% RSLogix 500 project FINAL PLC COMPLETE.RSS, saved by version 8.10.00.30 %
PROJECT "UNTITLED"    % processor: MicroLogix 1000 %

PROGRAM FILES
  LAD 2 "MAIN_PROG"  22 rungs
  LAD 3 "USER_FAULT"  1 rungs
  LAD 4 "HSC_INT"  1 rungs
  LAD 5 "STI_INT"  1 rungs
  LAD 6, 7, 8, 9, 10, 11, 12, 13, 14, 15, 16: only END

DATA FILES
  O0 OUTPUT  1 elements
  I1 INPUT  2 elements
  S2 STATUS  33 elements
  B3 BINARY  32 elements
  T4 TIMER  40 elements
  C5 COUNTER  32 elements
  R6 CONTROL  16 elements
  N7 INTEGER  105 elements

LADDER 2 "MAIN_PROG"
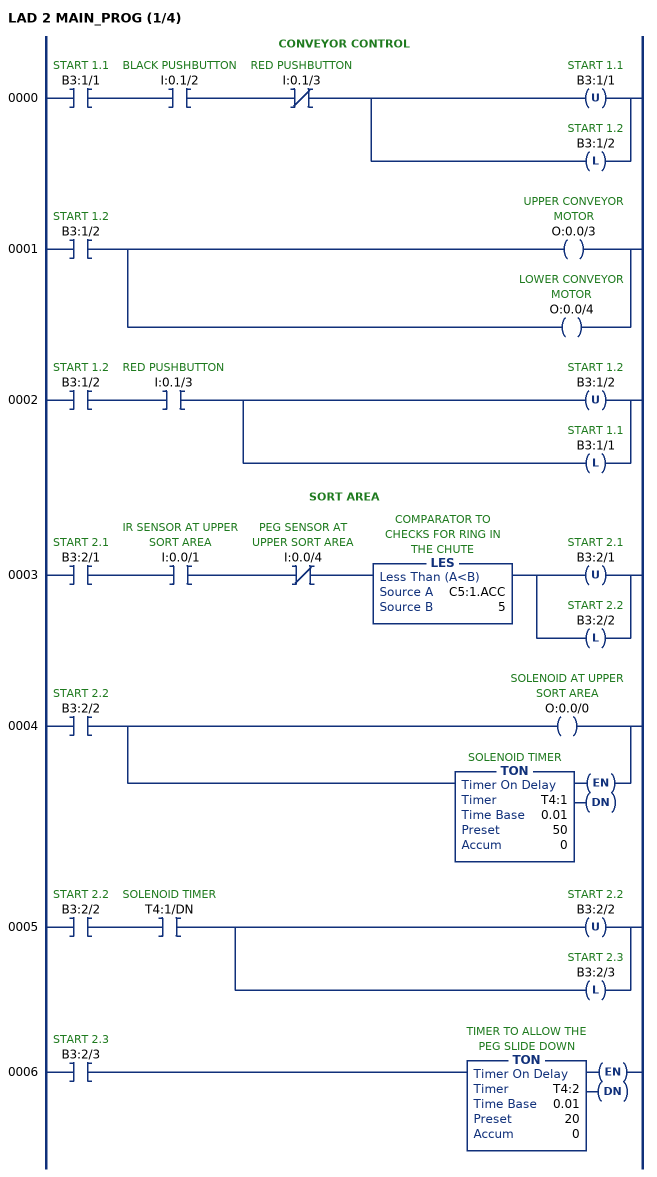
% Rung: 0 %
% TITLE: CONVEYOR CONTROL %
SOR XIC B3:1/1 XIC I:0.1/2 XIO I:0.1/3 BST OTU B3:1/1 NXB OTL B3:1/2 BND EOR
%   B3:1/1  "START 1.1" %
%   I:0.1/2  "BLACK PUSHBUTTON" %
%   I:0.1/3  "RED PUSHBUTTON" %
%   B3:1/2  "START 1.2" %
% Rung: 1 %
SOR XIC B3:1/2 BST OTE O:0.0/3 NXB OTE O:0.0/4 BND EOR
%   B3:1/2  "START 1.2" %
%   O:0.0/3  "UPPER CONVEYOR MOTOR" %
%   O:0.0/4  "LOWER CONVEYOR MOTOR" %
% Rung: 2 %
SOR XIC B3:1/2 XIC I:0.1/3 BST OTU B3:1/2 NXB OTL B3:1/1 BND EOR
%   B3:1/2  "START 1.2" %
%   I:0.1/3  "RED PUSHBUTTON" %
%   B3:1/1  "START 1.1" %
% Rung: 3 %
% TITLE: SORT AREA %
SOR XIC B3:2/1 XIC I:0.0/1 XIO I:0.0/4 LES C5:1.ACC 5 BST OTU B3:2/1 NXB OTL B3:2/2 BND EOR
%   B3:2/1  "START 2.1" %
%   I:0.0/1  "IR SENSOR AT UPPER SORT AREA" %
%   I:0.0/4  "PEG SENSOR AT UPPER SORT AREA" %
%   C5:1.ACC  "COMPARATOR TO CHECKS FOR RING IN THE CHUTE" %
%   B3:2/2  "START 2.2" %
% Rung: 4 %
SOR XIC B3:2/2 BST OTE O:0.0/0 NXB TON T4:1 0.01 50 0 BND EOR
%   B3:2/2  "START 2.2" %
%   O:0.0/0  "SOLENOID AT UPPER SORT AREA" %
%   T4:1  "SOLENOID TIMER" %
% Rung: 5 %
SOR XIC B3:2/2 XIC T4:1/DN BST OTU B3:2/2 NXB OTL B3:2/3 BND EOR
%   B3:2/2  "START 2.2" %
%   T4:1  "SOLENOID TIMER" %
%   B3:2/3  "START 2.3" %
% Rung: 6 %
SOR XIC B3:2/3 TON T4:2 0.01 20 0 EOR
%   B3:2/3  "START 2.3" %
%   T4:2  "TIMER TO ALLOW THE PEG SLIDE DOWN" %

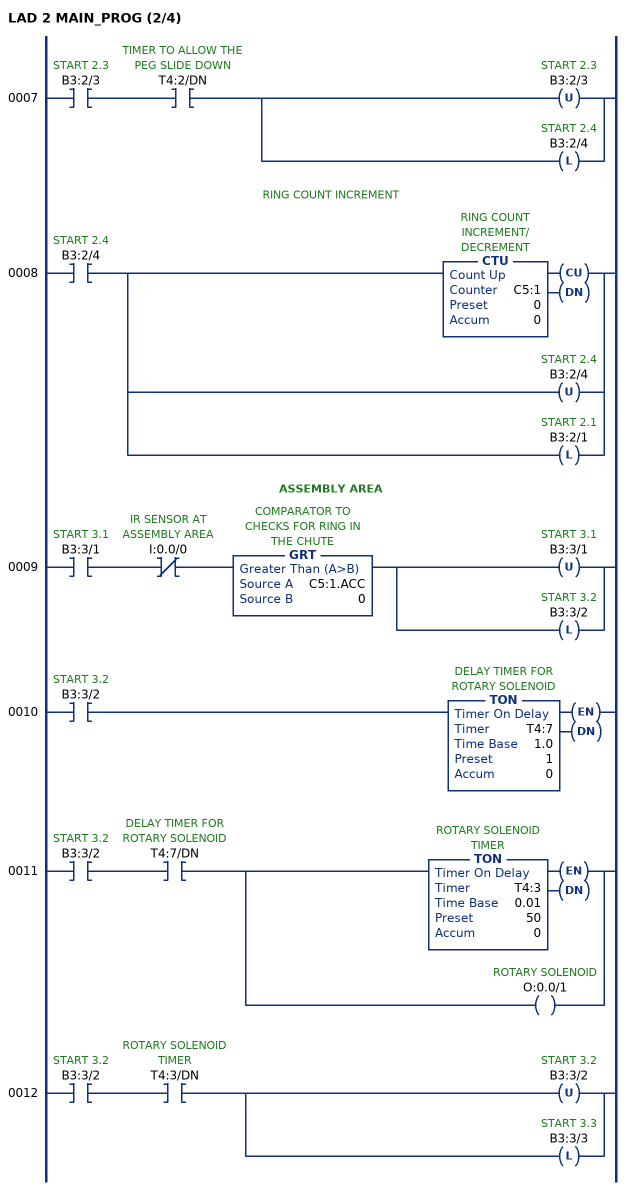
% Rung: 7 %
SOR XIC B3:2/3 XIC T4:2/DN BST OTU B3:2/3 NXB OTL B3:2/4 BND EOR
%   B3:2/3  "START 2.3" %
%   T4:2  "TIMER TO ALLOW THE PEG SLIDE DOWN" %
%   B3:2/4  "START 2.4" %
% Rung: 8 %
% RING COUNT INCREMENT %
SOR XIC B3:2/4 BST CTU C5:1 0 0 NXB BST OTU B3:2/4 NXB OTL B3:2/1 BND BND EOR
%   B3:2/4  "START 2.4" %
%   C5:1  "RING COUNT INCREMENT/DECREMENT" %
%   B3:2/1  "START 2.1" %
% Rung: 9 %
% TITLE: ASSEMBLY AREA %
SOR XIC B3:3/1 XIO I:0.0/0 GRT C5:1.ACC 0 BST OTU B3:3/1 NXB OTL B3:3/2 BND EOR
%   B3:3/1  "START 3.1" %
%   I:0.0/0  "IR SENSOR AT ASSEMBLY AREA" %
%   C5:1.ACC  "COMPARATOR TO CHECKS FOR RING IN THE CHUTE" %
%   B3:3/2  "START 3.2" %
% Rung: 10 %
SOR XIC B3:3/2 TON T4:7 1.0 1 0 EOR
%   B3:3/2  "START 3.2" %
%   T4:7  "DELAY TIMER FOR ROTARY SOLENOID" %
% Rung: 11 %
SOR XIC B3:3/2 XIC T4:7/DN BST TON T4:3 0.01 50 0 NXB OTE O:0.0/1 BND EOR
%   B3:3/2  "START 3.2" %
%   T4:7  "DELAY TIMER FOR ROTARY SOLENOID" %
%   T4:3  "ROTARY SOLENOID TIMER" %
%   O:0.0/1  "ROTARY SOLENOID" %
% Rung: 12 %
SOR XIC B3:3/2 XIC T4:3/DN BST OTU B3:3/2 NXB OTL B3:3/3 BND EOR
%   B3:3/2  "START 3.2" %
%   T4:3  "ROTARY SOLENOID TIMER" %
%   B3:3/3  "START 3.3" %

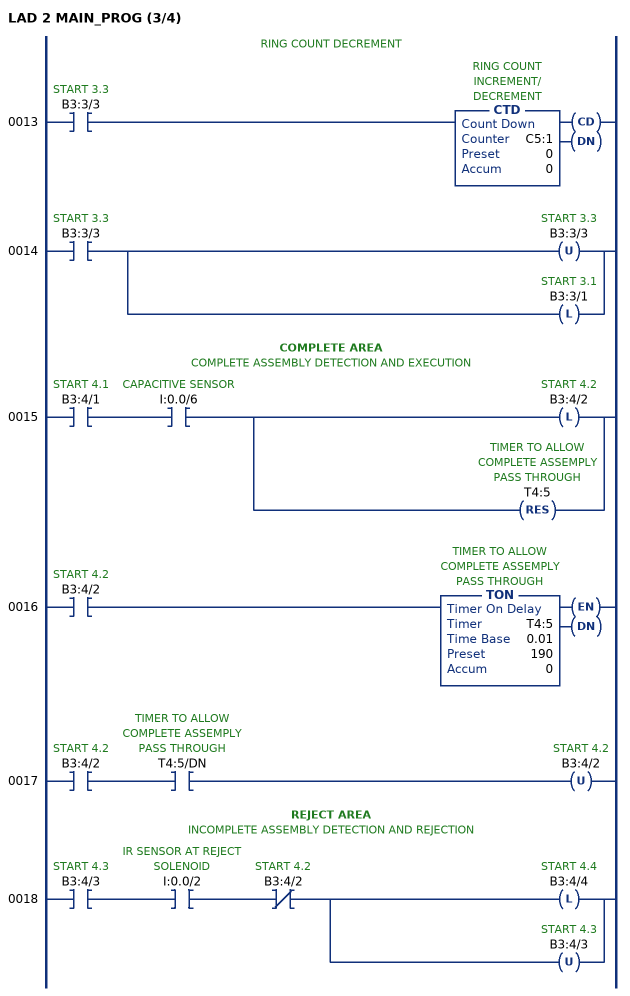
% Rung: 13 %
% RING COUNT DECREMENT %
SOR XIC B3:3/3 CTD C5:1 0 0 EOR
%   B3:3/3  "START 3.3" %
%   C5:1  "RING COUNT INCREMENT/DECREMENT" %
% Rung: 14 %
SOR XIC B3:3/3 BST OTU B3:3/3 NXB OTL B3:3/1 BND EOR
%   B3:3/3  "START 3.3" %
%   B3:3/1  "START 3.1" %
% Rung: 15 %
% TITLE: COMPLETE AREA %
% COMPLETE ASSEMBLY DETECTION AND EXECUTION %
SOR XIC B3:4/1 XIC I:0.0/6 BST OTL B3:4/2 NXB RES T4:5 BND EOR
%   B3:4/1  "START 4.1" %
%   I:0.0/6  "CAPACITIVE SENSOR" %
%   B3:4/2  "START 4.2" %
%   T4:5  "TIMER TO ALLOW COMPLETE ASSEMPLY PASS THROUGH" %
% Rung: 16 %
SOR XIC B3:4/2 TON T4:5 0.01 190 0 EOR
%   B3:4/2  "START 4.2" %
%   T4:5  "TIMER TO ALLOW COMPLETE ASSEMPLY PASS THROUGH" %
% Rung: 17 %
SOR XIC B3:4/2 XIC T4:5/DN OTU B3:4/2 EOR
%   B3:4/2  "START 4.2" %
%   T4:5  "TIMER TO ALLOW COMPLETE ASSEMPLY PASS THROUGH" %
% Rung: 18 %
% TITLE: REJECT AREA %
% INCOMPLETE ASSEMBLY DETECTION AND REJECTION %
SOR XIC B3:4/3 XIC I:0.0/2 XIO B3:4/2 BST OTL B3:4/4 NXB OTU B3:4/3 BND EOR
%   B3:4/3  "START 4.3" %
%   I:0.0/2  "IR SENSOR AT REJECT SOLENOID" %
%   B3:4/2  "START 4.2" %
%   B3:4/4  "START 4.4" %

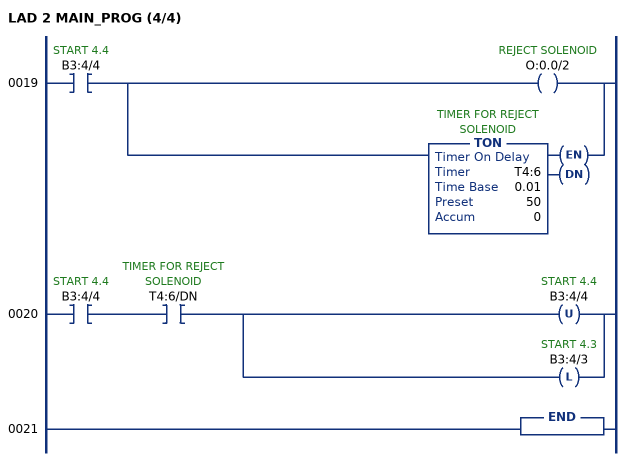
% Rung: 19 %
SOR XIC B3:4/4 BST OTE O:0.0/2 NXB TON T4:6 0.01 50 0 BND EOR
%   B3:4/4  "START 4.4" %
%   O:0.0/2  "REJECT SOLENOID" %
%   T4:6  "TIMER FOR REJECT SOLENOID" %
% Rung: 20 %
SOR XIC B3:4/4 XIC T4:6/DN BST OTU B3:4/4 NXB OTL B3:4/3 BND EOR
%   B3:4/4  "START 4.4" %
%   T4:6  "TIMER FOR REJECT SOLENOID" %
%   B3:4/3  "START 4.3" %
% Rung: 21 %
SOR END EOR

OTHER DOCUMENTED ADDRESSES
  B3:5/0  SW1  "START BUTTON ON SCADA"
  B3:5/1  SW2  "STOP BUTTON ON SCADA"
  B3:5/2  LED1
  B3:5/3  LED2

DATA TABLE (non-zero values as saved)
DATA B3
% B3:0 % 0X0000 0X0002 0X0002 0X000A 0X0012 0X0000 0X0000 0X0000 0X0000 0X0000
DATA T4
% .PRE .ACC %
% T4:1 % 50 0
% T4:2 % 20 0
% T4:3 % 50 0
% T4:4 % 50 0
% T4:5 % 190 0
% T4:6 % 50 0
% T4:7 % 1 0
